ADAPTER TokenRing (* Mutual Exclusion pattern adapter interface (dataless): RCV in, GIVE out *)
  (* Standard: 61499-1; Description: Copyright (c) 2026 HR Agrartechnik GmbH This program and the accompanying materials are made available under the terms of the Eclipse Public License 2.0 which is available at https://www.eclipse.org/legal/epl-2.0/ SPDX-License-Identifier: EPL-2.0 *)
  (* Version 1.1, 2026-08-31, Franz Höpfinger, HR Agrartechnik GmbH, GIVE/RCV Socket/Plug roles confirmed against the primary source: Dai/Vyatkin/Christensen/Dubinin, 'Function Block Implementation of Service Oriented Architecture: Case Study', IEEE INDIN 2014 - Section III.B: 'an adapter input MTXIN and output MTXOUT are reserved' *)
  (* Version 1.0, 2026-08-31, Franz Höpfinger, HR Agrartechnik GmbH, Mutual Exclusion / TokenRing design pattern (IEC 61499 primer course, Module 6, Valeriy Vyatkin, slide 15), initial version *)
  PACKAGE adapter::events::TokenRing;
  (* Documentation:
  Dataless adapter interface implementing the TokenRing / Mutual Exclusion design pattern (IEC 61499 primer course, Module 6, Valeriy Vyatkin, slide 15). Used to pass a mutual-exclusion "token" around a ring of controllers that share a resource: only the current token holder may enter its critical section; when done, it passes the token to its neighbour.
    - GIVE – from Plug to Socket: hand the token to the neighbour
   - RCV – from Socket to Plug: acknowledge that the token was received
    Plug (Name>>, named MTXOUT in the source) plays the "giver" role: fires GIVE, reacts to RCV. Socket (>>Name, named MTXIN) plays the "receiver" role: reacts to GIVE, fires RCV. A controller in the ring needs two instances - one MTXOUT (Plug) towards its downstream neighbour, one MTXIN (Socket) towards its upstream neighbour.
   Source: W. Dai, V. Vyatkin, J. H. Christensen, V. Dubinin, "Function Block Implementation of Service Oriented Architecture: Case Study," IEEE INDIN 2014, Section III.B/IV.A and Fig. 7/10 (local file INDIN14_DVCD.pdf) - confirms "an adapter input MTXIN and output MTXOUT are reserved" and that MTXIN/MTXOUT are wired into a ring to implement mutually exclusive access. See test_AX/Meins/DesingPatterns/TokenRingPattern/TokenRingPattern.md for the full write-up.
  *)
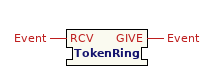
  EVENT_INPUT
    RCV; (* Acknowledgement from Socket that it received the token, sent back to Plug *)
  END_EVENT
  EVENT_OUTPUT
    GIVE; (* Plug hands the token to Socket *)
  END_EVENT
  SERVICE PLUG/SOCKET
    SEQUENCE token_pass
      PLUG.GIVE() -> SOCKET.GIVE();
      SOCKET.RCV() -> PLUG.RCV();
    END_SEQUENCE
  END_SERVICE
END_ADAPTER
